FUNCTION_BLOCK TEMPLATE_NEURALFB
  (* Standard: 61499-2 *)
  (* Version 1.0, 11-01-12, GASR, Universidade do Estado de Santa Catarina *)
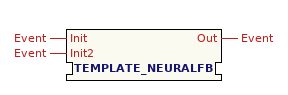
  EVENT_INPUT
    Init;
    Init2;
  END_EVENT
  EVENT_OUTPUT
    Out;
  END_EVENT
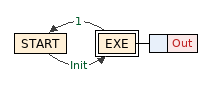
  EC_STATES
    EXE : -> Out;
    START;
  END_STATES
  EC_TRANSITIONS
    START TO EXE := Init;
    EXE TO START := 1;
  END_TRANSITIONS
END_FUNCTION_BLOCK
